{attribute 'GeneratedUsingTerminal: EP1122-0001-0016'}
{attribute addProperty BoxType "EP1122-0001-0016"}
{attribute addProperty Id "InfoDataAT %I*InfoData_6F19DB2B2"}
{attribute addProperty CRC "532711307"}
{attribute addProperty Size "2"}
TYPE EP1122_1FC0878B EXTENDS EtcSlaveTerminalBase_947E5A46 :
STRUCT
	{attribute addProperty Name "InfoData"}
	InfoData : InfoData_6F19DB2B;
END_STRUCT
END_TYPE

(* stored: Version 1.2.0.0, ProductVersion 3.1.4024.9
   DUT EP1122_1FC0878B: Id {8e4957a6-cf25-4f75-992c-405dc12f2e3f} *)
